Staubli VAL3: master1.pjx

Parameters version=s7.7.2 stackSize=5000 millimeterUnit=true
Program file=start.pgx
Program file=stop.pgx
Data file=master1.dtx
